TYPE EL6022_EX EXTENDS EL6022 :
STRUCT
	WcState AT %I* : BOOL;
	InputToggle AT %I* : BOOL;
	State AT %I* : UINT;
	AdsAdr AT %I* : Global.AMSADDR;
END_STRUCT
END_TYPE

(* stored: Version 1.1.0.1, ProductVersion 3.1.4026.18
   DUT EL6022_EX: Id {9fb93882-ca11-4e2e-ad6f-dc6ce40c84ca} *)
